{attribute 'GeneratedUsingTerminal: EL5002-0000-0020'}
{attribute addProperty BoxType "EL5002-0000-0020"}
{attribute addProperty Id "SSI_Inputs_Channel_1AT %I*SSI_Inputs_Channel_EDA1628411SSI_Inputs_Channel_2AT %I*SSI_Inputs_Channel_EDA1628411WcStateAT %I*WcState_9091E0EB2InfoDataAT %I*InfoData_94A18F5E2"}
{attribute addProperty CRC "1007138389"}
{attribute addProperty Size "26"}
TYPE EL5002_3C07B655 EXTENDS EtcSlaveTerminalBase_947E5A46 :
STRUCT
	{attribute addProperty Name "SSI_Inputs_Channel_1"}
	SSI_Inputs_Channel_1 : SSI_Inputs_Channel_EDA16284;
	{attribute addProperty Name "SSI_Inputs_Channel_2"}
	SSI_Inputs_Channel_2 : SSI_Inputs_Channel_EDA16284;
	{attribute addProperty Name "WcState"}
	WcState : WcState_9091E0EB;
	{attribute addProperty Name "InfoData"}
	InfoData : InfoData_94A18F5E;
END_STRUCT
END_TYPE

(* stored: Version 1.2.0.0, ProductVersion 3.1.4024.9
   DUT EL5002_3C07B655: Id {e41657ee-3444-42da-a640-803ddc70fde2} *)
